// TwinCAT 3 PLC project PLC
// ProgramVersion: 3.1.4024.0
// libraries:
//   Tc2_MC2, * (Beckhoff Automation GmbH)
//   Tc2_MC2_Drive, * (Beckhoff Automation GmbH)
//   Tc2_Standard, * (Beckhoff Automation GmbH)
//   Tc2_System, * (Beckhoff Automation GmbH)
//   Tc2_Utilities, * (Beckhoff Automation GmbH)
//   Tc3_Module, * (Beckhoff Automation GmbH)
// project tree:
//   DUTs/ ST_CSV_Record.TcDUT (not stored), st_driveControl.TcDUT
//   GVLs/ cabinet.TcGVL, driveController.TcGVL, GVL.TcGVL
//   / PlcTask.TcTTO
//   POUs/ button.TcPOU, drives.TcPOU, F.TcPOU, MAIN.TcPOU, P_TextModeWrite.TcPOU
// real-time tasks:
//   TASK PlcTask: cycle T#10ms, priority 20, ADS port 350
// motion (NC):
//   TASK NC-Task 1 SAF: cycle T#2ms, priority 4, ADS port 501
//   TASK NC-Task 1 SVB: cycle T#10ms, priority 8, ADS port 511
//   AXIS smallDrive (id 3)
//     Dynamic: Acceleration=5971.64, Deceleration=5971.64, Jerk=17914.9
//     Velo: RefSearch=39.8109354666667, RefSync=39.8109354666667, SlowManual=199.054677333333, FastManual=1194.328064, Fast=3981.09354666667, Maximum=3981.09
//     PositionAreaControl: Enable=false
//     TargetPosControl: Enable=false
//     OtherSettings: AllowMotionCmdToSlave=true
//     encoder EncType=19
//       EncPara: ScaleFactorNumerator=104.8576, ScaleFactorDenominator=1048576, MaxCount=#xffffffff
//     drive DrvType=16
//       DrvPara: MaxCount=#xffffffff, DriveControlDWord=#x00020000
//         Analog: VeloReferenz=4379.20290133333, VeloScale=32, TorqueSetpointScale=10, ScaleFactorActTorque=0.1
//         TimeComp: TaskDelayCycles=1
//     controller CtrType=1
//       CtrPara: PriorControlFactor=1
//         PosDiffControl: Enable=false
//         Observer: BandWidth=20
//   AXIS largeDrive (id 1)
//     PositionAreaControl: Enable=false
//     TargetPosControl: Enable=false
//     OtherSettings: AllowMotionCmdToSlave=true
//     encoder EncType=19
//       EncPara: MaxCount=#xffffffff
//     drive DrvType=16
//       DrvPara: MaxCount=#xffffffff, DriveControlDWord=#x00020000
//         Analog: TorqueSetpointScale=10, ScaleFactorActTorque=0.1
//         TimeComp: TaskDelayCycles=1
//     controller CtrType=1
//       CtrPara: PriorControlFactor=1
//         PosDiffControl: Enable=false
//         Observer: BandWidth=20
// I/O:
//   DEVICE Device 1 (EtherCAT), AmsNetId 192.168.2.188.2.1
//     Term 1 (EK1200) [EK1200-5000 EtherCAT Power supply (2A E-Bus)]
//       Term 2 (EL1809) [EL1809 16Ch. Dig. Input 24V, 3ms]
//       Term 3 (EL2809) [EL2809 16Ch. Dig. Output 24V, 0.5A]
//       Term 4 (EL3054) [EL3054 4Ch. Ana. Input 4-20mA]
//       Term 5 (EL4004) [EL4004 4Ch. Ana. Output 0-10V, 12bit]
//       Term 6 (EL9576) [EL9576 Brake chopper terminal]
//       Term 7 (EL7221-9014) [EL7221-9014 1Ch. MDP742 Servo motor output stage with OCT (50V, 8A RMS) and STO input]
//       Term 8 (EL7221-9014) [EL7221-9014 1Ch. MDP742 Servo motor output stage with OCT (50V, 8A RMS) and STO input]
//       Term 9 (EL1904) [EL1904, 4 Ch. Safety Input 24V, TwinSAFE]
//         modules: Module 1 (FSOES)
//       Term 10 (EL6021) [EL6021 Interface (RS422/485)]
//       Term 11 (EL9011) [EL9011 End Terminal]
// variable links:
//   NC-Task 1 SAF/Axes/largeDrive <-> Device 1 (EtherCAT)/Term 1 (EK1200)/Term 8 (EL7221-9014)
//     Drive/Inputs/In/nDcOutputTime <-> InfoData/DcOutputShift
//     Drive/Inputs/In/nState1 <-> DRV Statusword/Statusword
//     Drive/Inputs/In/nState2 <-> DRV Statusword/Statusword @bit 8
//     Drive/Inputs/In/nState4 @bit 1 <-> WcState/InputToggle
//     Drive/Inputs/In/nState4 <-> WcState/WcState
//     Drive/Outputs/Out/nCtrl1 <-> DRV Controlword/Controlword
//     Drive/Outputs/Out/nCtrl2 <-> DRV Controlword/Controlword @bit 8
//     Drive/Outputs/Out/nDataOut2 <-> DRV Target velocity/Target velocity
//     Enc/Inputs/In/nDataIn1 <-> FB Position/Position
//     Enc/Inputs/In/nDcInputTime <-> InfoData/DcInputShift
//     Enc/Inputs/In/nState4 @bit 1 <-> WcState/InputToggle
//     Enc/Inputs/In/nState4 <-> WcState/WcState
//   NC-Task 1 SAF/Axes/smallDrive <-> Device 1 (EtherCAT)/Term 1 (EK1200)/Term 7 (EL7221-9014)
//     Drive/Inputs/In/nDcOutputTime <-> InfoData/DcOutputShift
//     Drive/Inputs/In/nState1 <-> DRV Statusword/Statusword
//     Drive/Inputs/In/nState2 <-> DRV Statusword/Statusword @bit 8
//     Drive/Inputs/In/nState4 @bit 1 <-> WcState/InputToggle
//     Drive/Inputs/In/nState4 <-> WcState/WcState
//     Drive/Outputs/Out/nCtrl1 <-> DRV Controlword/Controlword
//     Drive/Outputs/Out/nCtrl2 <-> DRV Controlword/Controlword @bit 8
//     Drive/Outputs/Out/nDataOut2 <-> DRV Target velocity/Target velocity
//     Enc/Inputs/In/nDataIn1 <-> FB Position/Position
//     Enc/Inputs/In/nDcInputTime <-> InfoData/DcInputShift
//     Enc/Inputs/In/nState4 @bit 1 <-> WcState/InputToggle
//     Enc/Inputs/In/nState4 <-> WcState/WcState
//   PLC/PLC Instance <-> Device 1 (EtherCAT)/Term 1 (EK1200)/Term 2 (EL1809)
//     PlcTask Inputs/cabinet.emergencysw <-> Channel 7/Input
//     PlcTask Inputs/cabinet.motor1fwd <-> Channel 1/Input
//     PlcTask Inputs/cabinet.motor2fwd <-> Channel 3/Input
//     PlcTask Inputs/cabinet.motor1rev <-> Channel 2/Input
//     PlcTask Inputs/cabinet.motor2rev <-> Channel 4/Input
//     PlcTask Inputs/cabinet.selector1 <-> Channel 6/Input
//     PlcTask Inputs/cabinet.selector2 <-> Channel 5/Input
//   PLC/PLC Instance <-> Device 1 (EtherCAT)/Term 1 (EK1200)/Term 3 (EL2809)
//     PlcTask Outputs/cabinet.greenlight <-> Channel 2/Output
//     PlcTask Outputs/cabinet.orangelight <-> Channel 1/Output
//     PlcTask Outputs/cabinet.redlight <-> Channel 3/Output
//   PLC/PLC Instance <-> NC-Task 1 SAF/Axes/largeDrive
//     PlcTask Inputs/drives.alargeDrive.NcToPlc <-> Outputs/ToPlc
//     PlcTask Outputs/drives.alargeDrive.PlcToNc <-> Inputs/FromPlc
//   PLC/PLC Instance <-> NC-Task 1 SAF/Axes/smallDrive
//     PlcTask Inputs/drives.aSmallDrive.NcToPlc <-> Outputs/ToPlc
//     PlcTask Outputs/drives.aSmallDrive.PlcToNc <-> Inputs/FromPlc

CONFIGURATION PLC
    RESOURCE PLC ON TwinCAT3
        TASK PlcTask(INTERVAL := T#10ms, PRIORITY := 20);
        PROGRAM MAIN WITH PlcTask : MAIN;
    END_RESOURCE
END_CONFIGURATION

// ---- DUTs/st_driveControl.TcDUT
TYPE st_driveControl :
STRUCT
	
	xForward		: BOOL;
	xReverse		: BOOL;
	actualposition  : REAL;

END_STRUCT
END_TYPE

// ---- GVLs/cabinet.TcGVL
{attribute 'qualified_only'}
VAR_GLOBAL
	//INPUT 
	motor1fwd		AT %I*	: BOOL;
	motor1rev 		AT %I*	: BOOL;
	motor2fwd		AT %I*	: BOOL;
	motor2rev 		AT %I*	: BOOL;
	selector2		AT %I*	: BOOL;
	selector1       AT %I*  : BOOL;
	emergencysw		AT %I* 	: BOOL;
	
	//OUTPUT
	orangelight 	AT %Q*	: BOOL;
	greenlight		AT %Q*  : BOOL;
	redlight		AT %Q*  :BOOL;
	
	
	MAX_CSV_ROWS 			: UDINT := 100;
	MAX_CSV_COLUMNS 		: UDINT := 5;
	MAX_CSV_FIELD_LENGTH	: UDINT := 100;

END_VAR

// ---- GVLs/driveController.TcGVL
{attribute 'qualified_only'}
VAR_GLOBAL
	
	smallDrive			: st_driveControl;
    largeDrive      	: st_driveControl;
	
	largeacceleration 	: REAL;
	largevelocity		: REAL;
	largedeacceleration	: REAL;
	
	smallacceleration 	: REAL;
	smallvelocity		: REAL;
	smalldeacceleration	: REAL;
	
END_VAR

// ---- GVLs/GVL.TcGVL
VAR_GLOBAL CONSTANT
	MAX_CSV_ROWS 			: UDINT := 100;
	MAX_CSV_COLUMNS 		: UDINT := 5;
	MAX_CSV_FIELD_LENGTH	: UDINT := 100;
	
END_VAR

// ---- POUs/MAIN.TcPOU
PROGRAM MAIN
VAR

	bChangeSeparatorToComma: BOOL := FALSE;
END_VAR

IF bChangeSeparatorToComma THEN
	DEFAULT_CSV_FIELD_SEP := 16#2C;(* Comma ASCII code *)
ELSE
	DEFAULT_CSV_FIELD_SEP := 16#3B;(* Semicolon ASCII code *)
END_IF
P_TextModeWrite();

drives();
//F();e

END_PROGRAM

// ---- POUs/P_TextModeWrite.TcPOU
(* Writing of CSV file in text mode. None of the field value is containing any non-printing control characters like line feed, carriage return, quotation marks, semicolon... *)
PROGRAM P_TextModeWrite
VAR
	bWrite			: BOOL := FALSE;(* Rising edge starts program execution *)
	sNetId			: T_AmsNetId := '';	(* TwinCAT system network address *)
	sFileName		: T_MaxString := 'C:\CSV\TextModeGen.csv';(* CSV destination file path and name *)
	sCSVLine		: T_MaxString := '';(* Single CSV text line (row, record), we are using string as record buffer (your are able to see created fields) *)
	sCSVField		: T_MaxString := '';(* Single CSV field value (column, record field) *)
	bBusy			: BOOL;
	bError			: BOOL;
	nErrId			: UDINT;
	nRow	 		: UDINT 	:= 0;(* Row number (record) *)
	nColumn			: UDINT 	:= 0;(* Column number (record field) *)
	hFile			: UINT		:= 0;(* File handle of the source file *)
	step			: DWORD 	:= 0;
	fbFileOpen		: FB_FileOpen;(* Opens file *)
	fbFileClose		: FB_FileClose;(* Closes file *)
	fbFilePuts		: FB_FilePuts;(* Writes one record (line) *)
	fbWriter		: FB_CSVMemBufferWriter;(* Helper function block used to create CSV data bytes (single record line) *)

	database		: ARRAY[0..GVL.MAX_CSV_ROWS, 0..GVL.MAX_CSV_COLUMNS ] OF STRING(GVL.MAX_CSV_FIELD_LENGTH) :=[ (* Source PLC database *)
	'3_1', '0_1', '0_2', '0_3', '0_4', '0_5',
	'1_0', '1_1', '1_2', '1_3', '1_4', '1_5',
	'2_0', '2_1', '2_2', '2_3', '2_4', '2_5',
	'3_0', '3_1', '3_2', '3_3', '3_4', '3_5',
	'4_0', '4_1', '4_2', '4_3', '4_4', '4_5',
	'5_0', '5_1', '5_2', '5_3', '5_4', '5_5'];

END_VAR

CASE step OF
	0:	(* Wait for rising edge at bWrite variable *)
		IF bWrite THEN
			bWrite 	:= FALSE;
			bBusy 	:= TRUE;
			bError	:= FALSE;
			nErrId	:= 0;
			hFile	:= 0;
			nRow	:= 0;
			nColumn	:= 0;
			step 	:= 1;
		END_IF

	1:	(* Open source file *)
		fbFileOpen(  bExecute := FALSE  );
		fbFileOpen( sNetId := sNetId, sPathName := sFileName, nMode := FOPEN_MODEWRITE OR FOPEN_MODETEXT,(* Open file in TEXT mode! *)
					ePath := PATH_GENERIC, bExecute := TRUE );
		step := 2;

	2:(* Wait until open not busy *)
		fbFileOpen( bExecute := FALSE, bError => bError, nErrID => nErrID, hFile => hFile );
		IF NOT fbFileOpen.bBusy THEN
			IF NOT fbFileOpen.bError THEN
				step := 3;
			ELSE(* Error: file not found? *)
				step := 100;
			END_IF
		END_IF

	3:(* Convert one PLC record to CSV format *)
		sCSVLine := '';
		fbWriter.eCmd := eEnumCmd_First;(* Write first field value *)
		IF nRow <= GVL.MAX_CSV_ROWS THEN

			FOR nColumn := 0 TO GVL.MAX_CSV_COLUMNS BY 1 DO

				sCSVField := STRING_TO_CSVFIELD( database[ nRow, nColumn ], FALSE );(* TODO: Get field value from your application *)

				(* Add new field to the record buffer *)
				fbWriter( 	pBuffer := ADR( sCSVLine ), cbBuffer := SIZEOF( sCSVLine ) - 1, putValue := sCSVField, pValue := 0, cbValue := 0,
							bCRLF := ( nColumn = GVL.MAX_CSV_COLUMNS ) );(* bCRLF == TRUE => Write CRLF after the last field value *)
				IF fbWriter.bOk THEN
					fbWriter.eCmd := eEnumCmd_Next;(* Write next field value *)
				ELSE(* Error *)
					step := 100;
					RETURN;
				END_IF

			END_FOR(* FOR nColumn := 0... *)

			(* FB_FilePuts adds allready CR (carriage return) to the written line.
			We have to replace the $R$L characters with $L character to avoid double CR. *)
			IF RIGHT( sCSVLine, 2 ) = '$R$L' THEN
				sCSVLine := REPLACE( sCSVLine, '$L', 2, LEN( sCSVLine ) - 1 );
			END_IF

			nRow := nRow + 1;(* Increment number of created records (rows) *)
			step := 4;(* Write record to the file *)

		ELSE(* All rows written => Close file *)
			step := 10;
		END_IF

	4:	(* Write single text line *)
		fbFilePuts( bExecute := FALSE );
		fbFilePuts( sNetId := sNetId, hFile := hFile, sLine := sCSVLine, bExecute := TRUE );
		step := 5;

	5:(* Wait until write not busy *)
		fbFilePuts( bExecute := FALSE, bError => bError, nErrID => nErrID );
		IF NOT fbFilePuts.bBusy THEN
			IF NOT fbFilePuts.bError THEN
				step := 3;(* Write next record *)
			ELSE(* Error *)
				step := 100;
			END_IF
		END_IF

	10:	(* Close source file *)
		fbFileClose( bExecute := FALSE );
		fbFileClose( sNetId := sNetId, hFile := hFile, bExecute := TRUE );
		step := 11;

	11:(* Wait until close not busy *)
		fbFileClose( bExecute := FALSE, bError => bError, nErrID => nErrID );
		IF ( NOT fbFileClose.bBusy ) THEN
			hFile := 0;
			step := 100;
		END_IF

	100: (* Error or ready step => cleanup *)
		IF ( hFile <> 0 ) THEN
			step := 10; (* Close the source file *)
		ELSE
			bBusy := FALSE;
			step := 0;	(* Ready *)
		END_IF

END_CASE

END_PROGRAM

// ---- POUs/drives.TcPOU
PROGRAM drives
VAR
	//Small Drive
	aSmallDrive					: AXIS_REF; //initilization of asmallDrive axis
	MC_Power_aSmallDrive		: MC_Power; // linking to the FB
	MC_JOG_aSmallDrive			: MC_Jog;   //linking to the FB
	
	//LargeDrive
	alargeDrive					: AXIS_REF;	
	MC_Power_aLargeDrive		: MC_Power;
	MC_JOG_aLargeDrive			: MC_Jog;
	
	Read_Actual_position		: MC_ReadActualPosition;
	ActualPositionArrayLargeDrive 		: ARRAY [1..100000] OF REAL;
	ActualPositionArraysmallDrive 		: ARRAY [1..100000] OF REAL;
	Reset_largeDrive			: MC_Reset;
	Reset_smallDrive			: MC_Reset;
	
	Index 						: INT:=1; //Index of an array
	PositionlargeDrive					: REAL;	  //positoin variable initialisation
	PositionSmallDrive			:REAL;
    TIMER						: TON;    //FB link of TON
	
	{attribute 'OPC.UA.DA' := '1'}
	testVar						: BOOL;
	
	{attribute 'OPC.UA.DA' := '1'}
	testVar1					: BOOL;
	
	{attribute 'OPC.UA.DA' := '1'}
	testVar2					: BOOL;
	
	
	
	
	//variables set for motor config 
	largevelocity				: REAL;
	smallvelocity				: REAL;
	largedeacceleration			: REAL;
	largeacceleration			: REAL;
	smallacceleration			: REAL;
	smalldeacceleration			: REAL;
	
	//variables set for complete control 
	motor1fwdscada 				:BOOL;
	motor1revscada 				:BOOL;
	
	
	
	
	
	
END_VAR

//conditional statement for switching the RGB, Red for Emergency Stop , Green for motor 1 and Orange for motor2
IF NOT cabinet.emergencysw THEN
	Reset_largeDrive.Execute 			:= FALSE;
	Reset_smallDrive.Execute			:= FALSE;
    cabinet.redlight    				:= TRUE;
    cabinet.greenlight  				:= FALSE;
    cabinet.orangelight 				:= FALSE;
ELSIF cabinet.emergencysw AND cabinet.selector1 THEN
	Reset_smallDrive.Execute			:= TRUE;
    cabinet.redlight    				:= FALSE;
    cabinet.greenlight  				:= TRUE;
    cabinet.orangelight 				:= FALSE;   
ELSIF cabinet.emergencysw AND cabinet.selector2 THEN 
	Reset_largeDrive.Execute			:= TRUE;
    cabinet.redlight   					:= FALSE;
    cabinet.greenlight  				:= FALSE;
    cabinet.orangelight 				:= TRUE; 
END_IF

//Emergency switch to stop the motors
IF cabinet.emergencysw THEN
    drives.MC_Power_aSmallDrive.Enable := TRUE;
	drives.MC_Power_aLargeDrive.Enable := TRUE;
ELSE	
	drives.MC_Power_aSmallDrive.Enable := FALSE;
	drives.MC_Power_aLargeDrive.Enable := FALSE;
END_IF


////Selector conditonal statement
//IF cabinet.selector1 THEN
	
//	driveController.smallDrive.xForward := cabinet.motor1fwd;
//	driveController.smallDrive.xReverse := cabinet.motor1rev;
//ELSE
//	driveController.largeDrive.xForward := cabinet.motor2fwd;
//	driveController.largeDrive.xReverse := cabinet.motor2rev;	
//END_IF


WHILE cabinet.selector1 DO
	
	IF motor1fwdscada THEN
		driveController.smallDrive.xForward := TRUE;
	ELSIF motor1revscada THEN
		driveController.smallDrive.xReverse := TRUE;
		
	END_IF  
	
END_WHILE

//FB to read the positon of the large servo motor
Read_Actual_position(
	Axis								:= alargeDrive, 
	Enable								:= TRUE , 
	Valid=> , 
	Busy=> , 
	Error=> , 
	ErrorID=> , 
	Position							 => driveController.largeDrive.actualposition);
	

//FB to read the positon of the small servo motor
Read_Actual_position(
	Axis								:= asmallDrive, 
	Enable								:= TRUE , 
	Valid=> , 
	Busy=> , 
	Error=> , 
	ErrorID=> , 
	Position							 => driveController.smallDrive.actualposition);
	
//Fb to reset the large servo motor
Reset_largeDrive(
	Axis								:= alargeDrive, 
	Execute								:=  , 
	Done=> , 
	Busy=> , 
	Error=> , 
	ErrorID=> );

//FB to reset the small servo motor
Reset_smallDrive(
	Axis								:=aSmallDrive , 
	Execute								:= , 
	Done=> , 
	Busy=> , 
	Error=> , 
	ErrorID=> );
//seting up the defualt motor speed if velicty, acceleration and deacceleration is set to zero by user 

	IF driveController.largevelocity < 100 THEN
		largevelocity := 100.00;
	ELSE
		largevelocity := driveController.largevelocity;
	END_IF
	IF driveController.largeacceleration < 100 THEN
		largeacceleration:= 100.00;
	ELSE
		largeacceleration := driveController.largedeacceleration;
	END_IF
	IF driveController.largedeacceleration < 100 THEN
		largedeacceleration := 100.00;
	ELSE
		largedeacceleration := driveController.largedeacceleration;
	END_IF

	IF driveController.smallvelocity < 100 THEN
		smallvelocity := 100.00;
	ELSE
		smallvelocity := driveController.smallvelocity;
	END_IF
	IF driveController.smallacceleration < 100 THEN
		smallacceleration := 100.00;
	ELSE
		smallacceleration := driveController.smalldeacceleration;
	END_IF
	IF driveController.smalldeacceleration < 100 THEN
		smalldeacceleration := 100.00;
	ELSE
		smalldeacceleration := driveController.smalldeacceleration;
	END_IF
 
	
	////////////////////////////////////////////////


//small motor power and jog
MC_Power_aSmallDrive(
		Axis							:= aSmallDrive, 
		Enable							:= , 
		Enable_Positive					:= TRUE, 
		Enable_Negative					:= TRUE, 
		Override						:= 100, 
		BufferMode						:= , 
		Options							:= , 
		Status							=> , 
		Busy							=> , 
		Active							=> , 
		Error							=> , 
		ErrorID							=> );
	
MC_JOG_aSmallDrive(
		Axis							:= aSmallDrive, 
		JogForward						:= driveController.smallDrive.xForward, 
		JogBackwards					:= driveController.smallDrive.xReverse, 
		Mode							:= E_JogMode.MC_JOGMODE_CONTINOUS,
		Position						:= ,
		Velocity						:= smallvelocity, 
		Acceleration					:= smallacceleration, 
		Deceleration					:= smalldeacceleration, 
		Jerk							:= 15000, 
		Done							=> , 
		Busy							=> , 
		Active							=> , 
		CommandAborted					=> , 
		Error							=> , 
		ErrorID							=> );
	


//large drive Power and jog
MC_Power_aLargeDrive(
		Axis							:=alargeDrive , 
		Enable							:= , 
		Enable_Positive					:=TRUE , 
		Enable_Negative					:=TRUE , 
		Override						:=100 , 
		BufferMode						:= , 
		Options							:= , 
		Status							=> , 
		Busy							=> , 
		Active							=> , 
		Error							=> , 
		ErrorID							=> );
		
		
		
	

	MC_JOG_aLargeDrive(
		Axis							:= alargeDrive, 
		JogForward						:= driveController.largeDrive.xForward, 
		JogBackwards					:= driveController.largeDrive.xReverse, 
		Mode							:= E_JogMode.MC_JOGMODE_CONTINOUS,
		Position						:= ,
		Velocity						:= largevelocity, 
		Acceleration					:= largeacceleration,		
		Deceleration					:= largedeacceleration,
		Jerk							:= 1000, 
		Done							=> , 
		Busy							=> , 
		Active							=> , 
		CommandAborted					=> , 
		Error							=> , 
		ErrorID							=> );

		
//Timed storing of actual posiotn of  servo motor

TIMER(IN:= , PT:= T#1S , Q=> , ET=>  );		
IF driveController.largeDrive.xForward OR driveController.largeDrive.xReverse OR driveController.smallDrive.xForward OR driveController.smallDrive.xReverse THEN
	TIMER(IN := TRUE);
END_IF

IF TIMER.Q THEN
    PositionlargeDrive := driveController.largeDrive.actualposition;
	PositionSmallDrive := driveController.smallDrive.actualposition;
    ActualPositionArrayLargeDrive[Index] := PositionlargeDrive;
	ActualPositionArraysmallDrive[Index] := PositionSmallDrive;
	
    Index := Index + 1;
	Timer(IN := FALSE);
	
	
	IF Index > 100000 THEN
        Timer(IN := FALSE);  (* Stop the timer when 100000  values are stored *)
    END_IF
	
END_IF

END_PROGRAM

// ---- POUs/button.TcPOU
FUNCTION button : BOOL
VAR_INPUT
END_VAR
VAR
END_VAR

END_FUNCTION

// ---- POUs/F.TcPOU
PROGRAM F
VAR

	bWrite			: BOOL := FALSE;(* Rising edge starts program execution *)
	sNetId			: T_AmsNetId := '';	(* TwinCAT system network address *)
	sFileName		: T_MaxString := 'C:\CSV\yourfile.txt';(* CSV destination file path and name *)
	sCSVLine		: T_MaxString := '';(* Single CSV text line (row, record), we are using string as record buffer (your are able to see created fields) *)
	sCSVField		: T_MaxString := '';(* Single CSV field value (column, record field) *)
	bBusy			: BOOL;
	bError			: BOOL;
	nErrId			: UDINT;
	nRow	 		: UDINT 	:= 0;(* Row number (record) *)
	nColumn			: UDINT 	:= 0;(* Column number (record field) *)
	hFile			: UINT		:= 0;(* File handle of the source file *)
	step			: DWORD 	:= 0;
	
	(*database		: ARRAY[0..MAX_CSV_ROWS, 0..MAX_CSV_COLUMNS ] OF STRING(MAX_CSV_FIELD_LENGTH) :=[ (* Source PLC database *)
	'0_0', '0_1', '0_2', '0_3', '0_4', '0_5',
	'1_0', '1_1', '1_2', '1_3', '1_4', '1_5',
	'2_0', '2_1', '2_2', '2_3', '2_4', '2_5',
	'3_0', '3_1', '3_2', '3_3', '3_4', '3_5',
	'4_0', '4_1', '4_2', '4_3', '4_4', '4_5',
	'5_0', '5_1', '5_2', '5_3', '5_4', '5_5'];*)
	
	database : ARRAY[1..5] OF INT :=[1,2,3,4,5];
	
	FileOpen		: FB_FileOpen;(* Opens file *)
	FILEWRITE        :FB_FileWrite;
END_VAR



FileOpen( bExecute := FALSE  );
IF FileOpen THEN
	FileOpen( sNetId := sNetId, sPathName := sFileName, nMode := FOPEN_MODEWRITE OR FOPEN_MODEBINARY, (* Open file in BINARY mode! *)
					ePath := PATH_GENERIC, bExecute := TRUE );
END_IF 


FILEWRITE.bExecute := FALSE;
IF FILEWRITE.bExecute  THEN
	
	FILEWRITE( sNetId := sNetId, hFile := hFile, pWriteBuff := database, cbWriteLen := , bExecute := TRUE );
END_IF

END_PROGRAM
